TYPE ST_Property :
STRUCT
	b1,b2,b3 : BOOL;
	r1,r2,r3 : REAL;	
END_STRUCT
END_TYPE

(* stored: Version 1.1.0.1, ProductVersion 3.1.4024.12
   DUT ST_Property: Id {71d69592-d6db-4e35-a4a5-5e821f70c327} *)
